// TIA Portal V17 export
// export: Created 2025-03-05T08:03:15.303072Z, ExportSetting WithDefaults, DisplayName Totally Integrated Automation Portal, DisplayVersion V17 Update 8, DisplayName TIA Portal Openness, DisplayVersion V17 Update 8, DisplayName TIA Portal Version Control Interface, DisplayVersion V17, DisplayName SINAMICS Startdrive Advanced, DisplayVersion V17 SP2, DisplayName SINAMICS Startdrive G110M, G120, G120C, G120D, G120P, G115D, DisplayVersion V17 SP2, DisplayName SINAMICS Startdrive G130, G150, S120, S150, SINAMICS MV, S210, DisplayVersion V17 SP2, DisplayName STEP 7 Professional, DisplayVersion V17 Update 8, DisplayName SINUMERIK ONE STEP 7 Toolbox, DisplayVersion V17 Update 12, DisplayName SINUMERIK 840D sl STEP 7 Toolbox, DisplayVersion V17 Update 12, DisplayName STEP 7 Safety, DisplayVersion V17 Update 6, DisplayName WinCC Advanced, DisplayVersion V17 Update 8
FUNCTION_BLOCK "FB22502_STIRRER_CONTROL"   // FB22502, LAD
{ S7_Optimized_Access := 'FALSE' }
VERSION : 0.1
// stored: AutoNumber false, IsIECCheckEnabled false, SetENOAutomatically false, UDAEnableTagReadback false
   VAR_INPUT
      CONTROL_ON_DELAYED : Bool;   // Control On Delayed
      MOTOR_CONDITIONS : Bool;   // Motor Conditions
      MOTOR_STATUS_ERROR : Bool;   // Motor Status Error
      MOTOR_STATUS_ENABLE : Bool;   // Motor Status Enable
      MOTOR_STATUS_REACHED : Bool;   // Motor Status Reached
      START_MANUAL_REQUEST : Bool;   // Start Manual Request
      START_SEMI_REQUEST : Bool;   // Start Semi Request
      START_AUTO_REQUEST : Bool;   // Start Auto Request
      START_PROGRAM_REQUEST : Bool;   // Start Program Request
      STOP_MANUAL_REQUEST : Bool;   // Stop Manual Request
      STOP_SEMI_REQUEST : Bool;   // Stop Semi Request
      STOP_AUTO_REQUEST : Bool;   // Stop Auto Request
      STOP_PROGRAM_REQUEST : Bool;   // Stop Program Request
      MOTOR_ACTUAL_POSITION : DInt;   // Motor Actual Position
      MOTOR_ACTUAL_VELOCITY : DInt;   // Motor Actual Velocity
      MOTOR_ACTUAL_CURRENT : DInt;   // Motor Actual Current
      MOTOR_ACTUAL_CURRENT_FILTERED : DInt;   // Motor Actual Current Filtered
      MOTOR_ACTUAL_TEMPERATURE : Real;   // Motor Actual Temperature
      MOTOR_STATUS_REGISTER : UDInt;   // Motor Status Register
   END_VAR
   VAR_OUTPUT
      "MOTOR _VELOCITY _TARGET _SOURCE" : DInt;   // MOTOR VELOCITY TARGET SOURCE
      "MOTOR _MODE _OF _OPERATION" : Int;   // MOTOR MODE OF OPERATION
      "MOTOR _ENABLE _POWER _STAGE" : Int;   // MOTOR ENABLE POWER STAGE
      "MOTOR _OUT1" : Bool;   // MOTOR OUT1
      "MOTOR _OUT2" : Bool;   // MOTOR OUT2
      "MOTOR _OUT3" : Bool;   // MOTOR OUT3
      "MOTOR _ENABLE _1" : Bool;   // MOTOR ENABLE 1
      "MOTOR _ENABLE _2" : Bool;   // MOTOR ENABLE 2
      "CURRENT _LIMIT _ALARM" : Bool;   // CURRENT LIMIT ALARM
      "TEMPRETATURE _LIMIT _ALARM" : Bool;   // TEMPRETATURE LIMIT ALARM
   END_VAR
   VAR DB_SPECIFIC
      DATA_STANDARD : "GENERAL_DATA_START_STOP";
      DATA_HMI : "HMI_DATA_START_STOP";
      INPUT_SETTINGS : Struct
         UNIT_NUMBER : Int;
         HOPPER_NUMBER : Int;
      END_STRUCT;
      ALARM_SETTINGS : Struct
         CURRENT_LIMIT : DInt;   // CURRENT LIMIT
         TEMPERATURE_LIMIT : Real;   // TEMPERATURE LIMIT
         TIMER_CURRENT_LIMIT : TON_TIME;   // TIMER CURRENT LIMIT
         TIMER_TEMPERATURE_LIMIT : TON_TIME;
      END_STRUCT;
      "HMI _SETPOINT _VELOCITY" : DInt;   // HMI SETPOINT VELOCITY
      "HMI _ACTUAL _POSITION" : DInt;   // HMI ACTUAL POSITION
      "HMI _ACTUAL _VELOCITY" : DInt;   // HMI ACTUAL VELOCITY
      "HMI _ACTUAL _CURRENT" : DInt;   // HMI ACTUAL CURRENT
      "HMI _ACTUAL _CURRENT _FILTERED" : DInt;   // HMI ACTUAL CURRENT FILTERED
      "HMI _STIRRER _LOW _RANGE" : DInt;   // HMI STIRRER LOW RANGE
      "HMI _STIRRER _HIGH _RANGE" : DInt;   // HMI STIRRER HIGH RANGE
      "PROGRAM _SETPOINT _VELOCITY" : DInt;   // PROGRAM SETPOINT VELOCITY
      "SETPOINT _VELOCITY" : DInt;   // SETPOINT VELOCITY
      "FEEDBACK _POSITION" : DInt;   // FEEDBACK POSITION
      "FEEDBACK _VELOCITY" : DInt;   // FEEDBACK VELOCITY
      "FEEDBACK _CURRENT" : DInt;   // FEEDBACK CURRENT
      "FEEDBACK _CURRENT _FILTERED" : DInt;   // FEEDBACK CURRENT FILTERED
      "FEEDBACK _TEMPERATURE" : Real;   // FEEDBACK TEMPERATURE
   END_VAR
   VAR_TEMP
      DB_NUMBER : DInt;
      RETVAL : Int;
   END_VAR
   // ALARM_SETTINGS.TIMER_CURRENT_LIMIT.PT := T#1s;
   // ALARM_SETTINGS.TIMER_TEMPERATURE_LIMIT.PT := T#1s;
   VAR_TEMP   // added for the SCL form of the ladder/FBD networks
      _w1 : Bool;
      _w2 : Bool;
   END_VAR
BEGIN

NETWORK
TITLE = READ INSTANCE DB NUMBER
      L     DINO;
      +     10#800000;
      T     #DB_NUMBER;


REGION Network 2: INPUTS
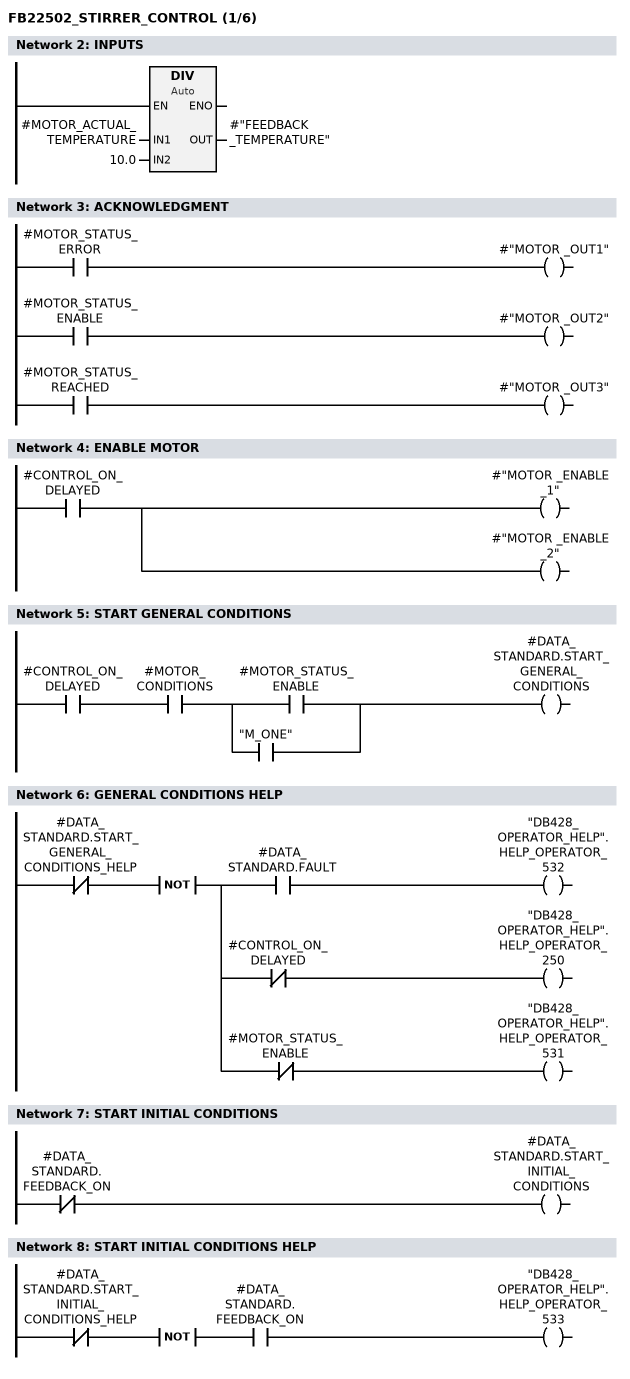
   RUNG wire#powerrail
      Div(in1 := #MOTOR_ACTUAL_TEMPERATURE, in2 := 10.0, out => #"FEEDBACK _TEMPERATURE")
   END_RUNG
   // the same network as SCL:
   #"FEEDBACK _TEMPERATURE" := #MOTOR_ACTUAL_TEMPERATURE / 10.0;
END_REGION

REGION Network 3: ACKNOWLEDGMENT
   RUNG wire#powerrail
      Contact( #MOTOR_STATUS_ERROR )
      Coil( #"MOTOR _OUT1" )
   END_RUNG
   RUNG wire#powerrail
      Contact( #MOTOR_STATUS_ENABLE )
      Coil( #"MOTOR _OUT2" )
   END_RUNG
   RUNG wire#powerrail
      Contact( #MOTOR_STATUS_REACHED )
      Coil( #"MOTOR _OUT3" )
   END_RUNG
   // the same network as SCL:
   #"MOTOR _OUT1" := #MOTOR_STATUS_ERROR;
   #"MOTOR _OUT2" := #MOTOR_STATUS_ENABLE;
   #"MOTOR _OUT3" := #MOTOR_STATUS_REACHED;
END_REGION

REGION Network 4: ENABLE MOTOR
   RUNG wire#powerrail
      Contact( #CONTROL_ON_DELAYED )
      wire#w1
      Coil( #"MOTOR _ENABLE _1" )
   END_RUNG
   RUNG wire#w1
      Coil( #"MOTOR _ENABLE _2" )
   END_RUNG
   // the same network as SCL:
   #"MOTOR _ENABLE _1" := #CONTROL_ON_DELAYED;
   #"MOTOR _ENABLE _2" := #CONTROL_ON_DELAYED;
END_REGION

REGION Network 5: START GENERAL CONDITIONS
   RUNG wire#powerrail
      Contact( #CONTROL_ON_DELAYED )
      Contact( #MOTOR_CONDITIONS )
      wire#w1
      Contact( #MOTOR_STATUS_ENABLE )
      wire#w2
      Coil( #DATA_STANDARD.START_GENERAL_CONDITIONS )
   END_RUNG
   RUNG wire#w1
      Contact( "M_ONE" )
   END_RUNG wire#w2
   // the same network as SCL:
   #DATA_STANDARD.START_GENERAL_CONDITIONS := #CONTROL_ON_DELAYED AND #MOTOR_CONDITIONS AND (#MOTOR_STATUS_ENABLE OR "M_ONE");
END_REGION

REGION Network 6: GENERAL CONDITIONS HELP
   RUNG wire#powerrail
      I_Contact( #DATA_STANDARD.START_GENERAL_CONDITIONS_HELP )
      Not()
      wire#w1
      Contact( #DATA_STANDARD.FAULT )
      Coil( "DB428_OPERATOR_HELP".HELP_OPERATOR_532 )
   END_RUNG
   RUNG wire#w1
      I_Contact( #CONTROL_ON_DELAYED )
      Coil( "DB428_OPERATOR_HELP".HELP_OPERATOR_250 )
   END_RUNG
   RUNG wire#w1
      I_Contact( #MOTOR_STATUS_ENABLE )
      Coil( "DB428_OPERATOR_HELP".HELP_OPERATOR_531 )
   END_RUNG
   // the same network as SCL:
   #_w1 := NOT (NOT #DATA_STANDARD.START_GENERAL_CONDITIONS_HELP);
   "DB428_OPERATOR_HELP".HELP_OPERATOR_532 := #_w1 AND #DATA_STANDARD.FAULT;
   "DB428_OPERATOR_HELP".HELP_OPERATOR_250 := #_w1 AND NOT #CONTROL_ON_DELAYED;
   "DB428_OPERATOR_HELP".HELP_OPERATOR_531 := #_w1 AND NOT #MOTOR_STATUS_ENABLE;
END_REGION

REGION Network 7: START INITIAL CONDITIONS
   RUNG wire#powerrail
      I_Contact( #DATA_STANDARD.FEEDBACK_ON )
      Coil( #DATA_STANDARD.START_INITIAL_CONDITIONS )
   END_RUNG
   // the same network as SCL:
   #DATA_STANDARD.START_INITIAL_CONDITIONS := NOT #DATA_STANDARD.FEEDBACK_ON;
END_REGION

REGION Network 8: START INITIAL CONDITIONS HELP
   RUNG wire#powerrail
      I_Contact( #DATA_STANDARD.START_INITIAL_CONDITIONS_HELP )
      Not()
      Contact( #DATA_STANDARD.FEEDBACK_ON )
      Coil( "DB428_OPERATOR_HELP".HELP_OPERATOR_533 )
   END_RUNG
   // the same network as SCL:
   "DB428_OPERATOR_HELP".HELP_OPERATOR_533 := NOT (NOT #DATA_STANDARD.START_INITIAL_CONDITIONS_HELP) AND #DATA_STANDARD.FEEDBACK_ON;
END_REGION

REGION Network 9: START MANUAL REQUEST
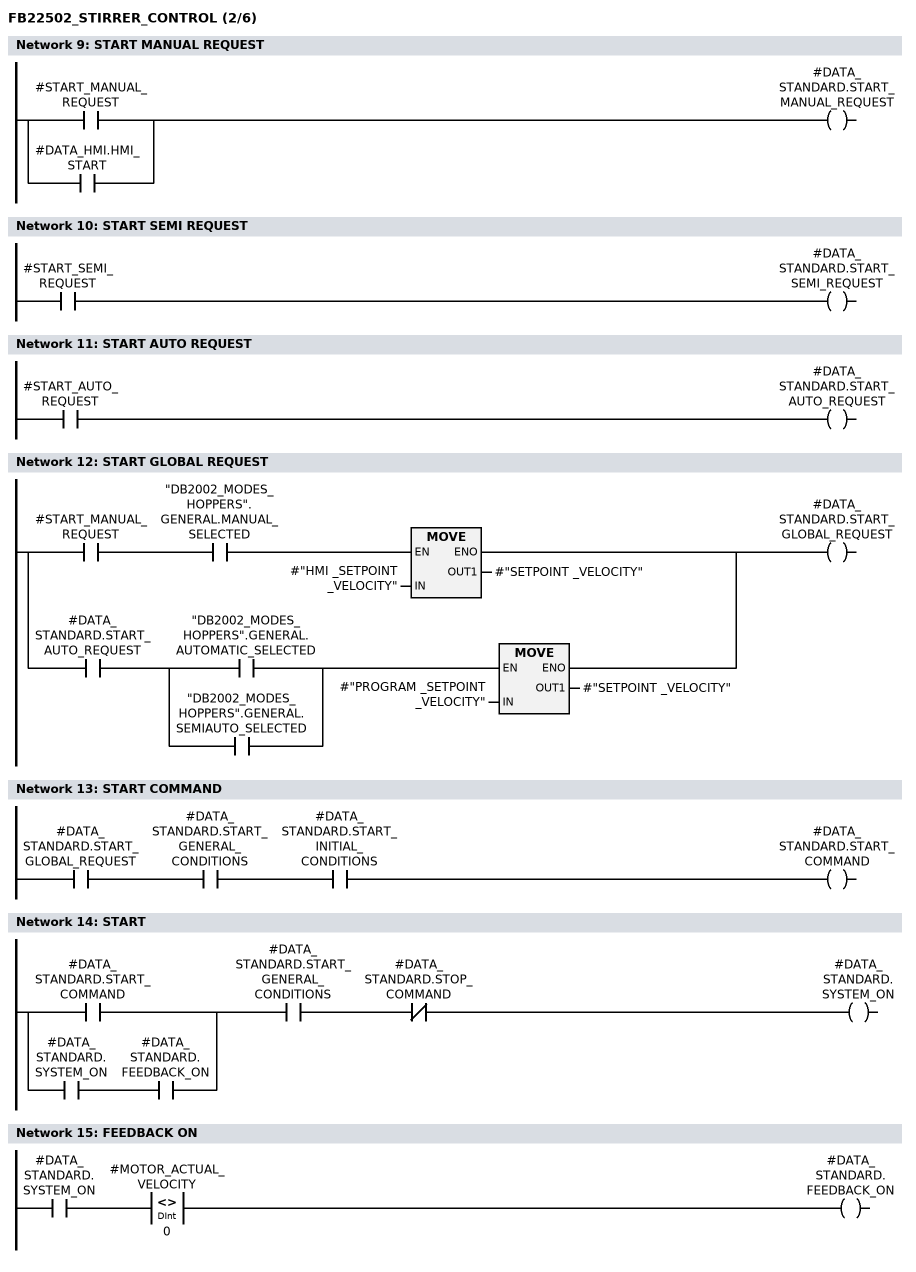
   RUNG wire#powerrail
      Contact( #START_MANUAL_REQUEST )
      wire#w1
      Coil( #DATA_STANDARD.START_MANUAL_REQUEST )
   END_RUNG
   RUNG wire#powerrail
      Contact( #DATA_HMI.HMI_START )
   END_RUNG wire#w1
   // the same network as SCL:
   #DATA_STANDARD.START_MANUAL_REQUEST := #START_MANUAL_REQUEST OR #DATA_HMI.HMI_START;
END_REGION

REGION Network 10: START SEMI REQUEST
   RUNG wire#powerrail
      Contact( #START_SEMI_REQUEST )
      Coil( #DATA_STANDARD.START_SEMI_REQUEST )
   END_RUNG
   // the same network as SCL:
   #DATA_STANDARD.START_SEMI_REQUEST := #START_SEMI_REQUEST;
END_REGION

REGION Network 11: START AUTO REQUEST
   RUNG wire#powerrail
      Contact( #START_AUTO_REQUEST )
      Coil( #DATA_STANDARD.START_AUTO_REQUEST )
   END_RUNG
   // the same network as SCL:
   #DATA_STANDARD.START_AUTO_REQUEST := #START_AUTO_REQUEST;
END_REGION

REGION Network 12: START GLOBAL REQUEST
   RUNG wire#powerrail
      Contact( #START_MANUAL_REQUEST )
      Contact( "DB2002_MODES_HOPPERS".GENERAL.MANUAL_SELECTED )
      Move(in := #"HMI _SETPOINT _VELOCITY", out1 => #"SETPOINT _VELOCITY")
      wire#w1
      Coil( #DATA_STANDARD.START_GLOBAL_REQUEST )
   END_RUNG
   RUNG wire#powerrail
      Contact( #DATA_STANDARD.START_AUTO_REQUEST )
      wire#w2
      Contact( "DB2002_MODES_HOPPERS".GENERAL.AUTOMATIC_SELECTED )
      wire#w3
      Move(in := #"PROGRAM _SETPOINT _VELOCITY", out1 => #"SETPOINT _VELOCITY")
   END_RUNG wire#w1
   RUNG wire#w2
      Contact( "DB2002_MODES_HOPPERS".GENERAL.SEMIAUTO_SELECTED )
   END_RUNG wire#w3
   // the same network as SCL:
   #_w1 := #START_MANUAL_REQUEST AND "DB2002_MODES_HOPPERS".GENERAL.MANUAL_SELECTED;
   IF #_w1 THEN #"SETPOINT _VELOCITY" := #"HMI _SETPOINT _VELOCITY"; END_IF;
   #_w2 := #DATA_STANDARD.START_AUTO_REQUEST AND ("DB2002_MODES_HOPPERS".GENERAL.AUTOMATIC_SELECTED OR "DB2002_MODES_HOPPERS".GENERAL.SEMIAUTO_SELECTED);
   IF #_w2 THEN #"SETPOINT _VELOCITY" := #"PROGRAM _SETPOINT _VELOCITY"; END_IF;
   #DATA_STANDARD.START_GLOBAL_REQUEST := #_w1 OR #_w2;
END_REGION

REGION Network 13: START COMMAND
   RUNG wire#powerrail
      Contact( #DATA_STANDARD.START_GLOBAL_REQUEST )
      Contact( #DATA_STANDARD.START_GENERAL_CONDITIONS )
      Contact( #DATA_STANDARD.START_INITIAL_CONDITIONS )
      Coil( #DATA_STANDARD.START_COMMAND )
   END_RUNG
   // the same network as SCL:
   #DATA_STANDARD.START_COMMAND := #DATA_STANDARD.START_GLOBAL_REQUEST AND #DATA_STANDARD.START_GENERAL_CONDITIONS AND #DATA_STANDARD.START_INITIAL_CONDITIONS;
END_REGION

REGION Network 14: START
   RUNG wire#powerrail
      Contact( #DATA_STANDARD.START_COMMAND )
      wire#w1
      Contact( #DATA_STANDARD.START_GENERAL_CONDITIONS )
      I_Contact( #DATA_STANDARD.STOP_COMMAND )
      Coil( #DATA_STANDARD.SYSTEM_ON )
   END_RUNG
   RUNG wire#powerrail
      Contact( #DATA_STANDARD.SYSTEM_ON )
      Contact( #DATA_STANDARD.FEEDBACK_ON )
   END_RUNG wire#w1
   // the same network as SCL:
   #DATA_STANDARD.SYSTEM_ON := (#DATA_STANDARD.START_COMMAND OR (#DATA_STANDARD.SYSTEM_ON AND #DATA_STANDARD.FEEDBACK_ON)) AND #DATA_STANDARD.START_GENERAL_CONDITIONS AND NOT #DATA_STANDARD.STOP_COMMAND;
END_REGION

REGION Network 15: FEEDBACK ON
   RUNG wire#powerrail
      Contact( #DATA_STANDARD.SYSTEM_ON )
      { S7_Templates := "SrcType := DInt" } NE_Contact(in1 := #MOTOR_ACTUAL_VELOCITY, in2 := 0)
      Coil( #DATA_STANDARD.FEEDBACK_ON )
   END_RUNG
   // the same network as SCL:
   #DATA_STANDARD.FEEDBACK_ON := #DATA_STANDARD.SYSTEM_ON AND (#MOTOR_ACTUAL_VELOCITY <> 0);
END_REGION

REGION Network 16: STOP GENERAL CONDITIONS
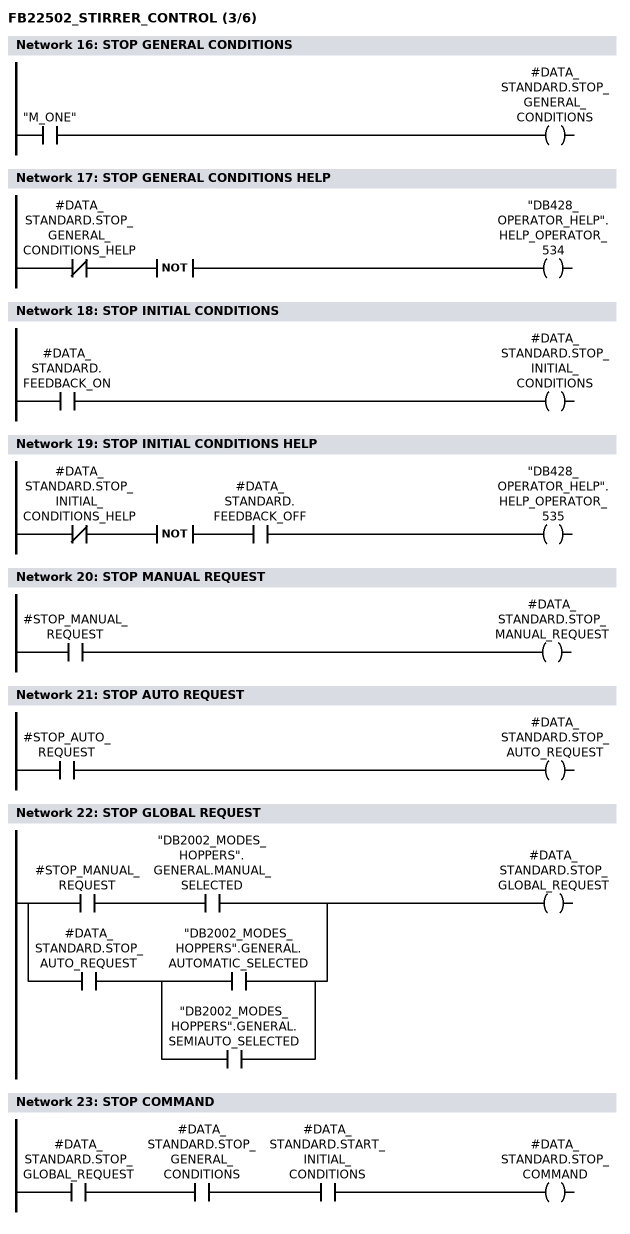
   RUNG wire#powerrail
      Contact( "M_ONE" )
      Coil( #DATA_STANDARD.STOP_GENERAL_CONDITIONS )
   END_RUNG
   // the same network as SCL:
   #DATA_STANDARD.STOP_GENERAL_CONDITIONS := "M_ONE";
END_REGION

REGION Network 17: STOP GENERAL CONDITIONS HELP
   RUNG wire#powerrail
      I_Contact( #DATA_STANDARD.STOP_GENERAL_CONDITIONS_HELP )
      Not()
      Coil( "DB428_OPERATOR_HELP".HELP_OPERATOR_534 )
   END_RUNG
   // the same network as SCL:
   "DB428_OPERATOR_HELP".HELP_OPERATOR_534 := NOT (NOT #DATA_STANDARD.STOP_GENERAL_CONDITIONS_HELP);
END_REGION

REGION Network 18: STOP INITIAL CONDITIONS
   RUNG wire#powerrail
      Contact( #DATA_STANDARD.FEEDBACK_ON )
      Coil( #DATA_STANDARD.STOP_INITIAL_CONDITIONS )
   END_RUNG
   // the same network as SCL:
   #DATA_STANDARD.STOP_INITIAL_CONDITIONS := #DATA_STANDARD.FEEDBACK_ON;
END_REGION

REGION Network 19: STOP INITIAL CONDITIONS HELP
   RUNG wire#powerrail
      I_Contact( #DATA_STANDARD.STOP_INITIAL_CONDITIONS_HELP )
      Not()
      Contact( #DATA_STANDARD.FEEDBACK_OFF )
      Coil( "DB428_OPERATOR_HELP".HELP_OPERATOR_535 )
   END_RUNG
   // the same network as SCL:
   "DB428_OPERATOR_HELP".HELP_OPERATOR_535 := NOT (NOT #DATA_STANDARD.STOP_INITIAL_CONDITIONS_HELP) AND #DATA_STANDARD.FEEDBACK_OFF;
END_REGION

REGION Network 20: STOP MANUAL REQUEST
   RUNG wire#powerrail
      Contact( #STOP_MANUAL_REQUEST )
      Coil( #DATA_STANDARD.STOP_MANUAL_REQUEST )
   END_RUNG
   // the same network as SCL:
   #DATA_STANDARD.STOP_MANUAL_REQUEST := #STOP_MANUAL_REQUEST;
END_REGION

REGION Network 21: STOP AUTO REQUEST
   RUNG wire#powerrail
      Contact( #STOP_AUTO_REQUEST )
      Coil( #DATA_STANDARD.STOP_AUTO_REQUEST )
   END_RUNG
   // the same network as SCL:
   #DATA_STANDARD.STOP_AUTO_REQUEST := #STOP_AUTO_REQUEST;
END_REGION

REGION Network 22: STOP GLOBAL REQUEST
   RUNG wire#powerrail
      Contact( #STOP_MANUAL_REQUEST )
      Contact( "DB2002_MODES_HOPPERS".GENERAL.MANUAL_SELECTED )
      wire#w1
      Coil( #DATA_STANDARD.STOP_GLOBAL_REQUEST )
   END_RUNG
   RUNG wire#powerrail
      Contact( #DATA_STANDARD.STOP_AUTO_REQUEST )
      wire#w2
      Contact( "DB2002_MODES_HOPPERS".GENERAL.AUTOMATIC_SELECTED )
   END_RUNG wire#w1
   RUNG wire#w2
      Contact( "DB2002_MODES_HOPPERS".GENERAL.SEMIAUTO_SELECTED )
   END_RUNG wire#w1
   // the same network as SCL:
   #DATA_STANDARD.STOP_GLOBAL_REQUEST := (#STOP_MANUAL_REQUEST AND "DB2002_MODES_HOPPERS".GENERAL.MANUAL_SELECTED) OR (#DATA_STANDARD.STOP_AUTO_REQUEST AND ("DB2002_MODES_HOPPERS".GENERAL.AUTOMATIC_SELECTED OR "DB2002_MODES_HOPPERS".GENERAL.SEMIAUTO_SELECTED));
END_REGION

REGION Network 23: STOP COMMAND
   RUNG wire#powerrail
      Contact( #DATA_STANDARD.STOP_GLOBAL_REQUEST )
      Contact( #DATA_STANDARD.STOP_GENERAL_CONDITIONS )
      Contact( #DATA_STANDARD.START_INITIAL_CONDITIONS )
      Coil( #DATA_STANDARD.STOP_COMMAND )
   END_RUNG
   // the same network as SCL:
   #DATA_STANDARD.STOP_COMMAND := #DATA_STANDARD.STOP_GLOBAL_REQUEST AND #DATA_STANDARD.STOP_GENERAL_CONDITIONS AND #DATA_STANDARD.START_INITIAL_CONDITIONS;
END_REGION

REGION Network 24: STOP
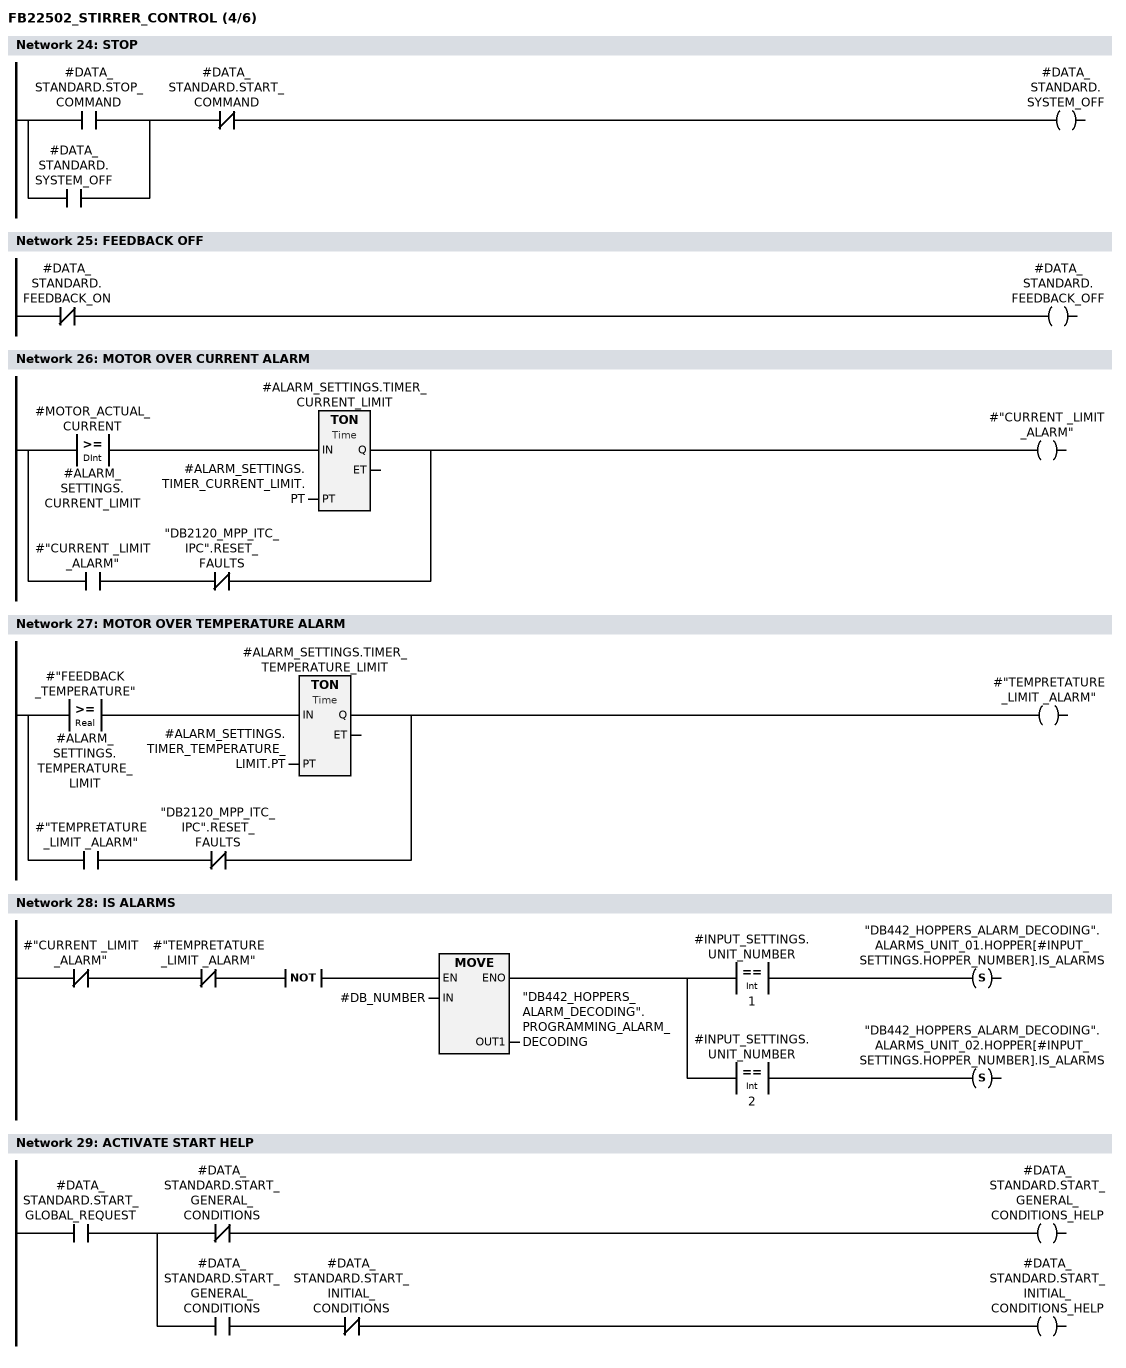
   RUNG wire#powerrail
      Contact( #DATA_STANDARD.STOP_COMMAND )
      wire#w1
      I_Contact( #DATA_STANDARD.START_COMMAND )
      Coil( #DATA_STANDARD.SYSTEM_OFF )
   END_RUNG
   RUNG wire#powerrail
      Contact( #DATA_STANDARD.SYSTEM_OFF )
   END_RUNG wire#w1
   // the same network as SCL:
   #DATA_STANDARD.SYSTEM_OFF := (#DATA_STANDARD.STOP_COMMAND OR #DATA_STANDARD.SYSTEM_OFF) AND NOT #DATA_STANDARD.START_COMMAND;
END_REGION

REGION Network 25: FEEDBACK OFF
   RUNG wire#powerrail
      I_Contact( #DATA_STANDARD.FEEDBACK_ON )
      Coil( #DATA_STANDARD.FEEDBACK_OFF )
   END_RUNG
   // the same network as SCL:
   #DATA_STANDARD.FEEDBACK_OFF := NOT #DATA_STANDARD.FEEDBACK_ON;
END_REGION

REGION Network 26: MOTOR OVER CURRENT ALARM
   RUNG wire#powerrail
      { S7_Templates := "SrcType := DInt" } GE_Contact(in1 := #MOTOR_ACTUAL_CURRENT, in2 := #ALARM_SETTINGS.CURRENT_LIMIT)
      { S7_Templates := "time_type := Time" } #ALARM_SETTINGS.TIMER_CURRENT_LIMIT.TON(pt := #ALARM_SETTINGS.TIMER_CURRENT_LIMIT.PT, et =>)
      wire#w1
      Coil( #"CURRENT _LIMIT _ALARM" )
   END_RUNG
   RUNG wire#powerrail
      Contact( #"CURRENT _LIMIT _ALARM" )
      I_Contact( "DB2120_MPP_ITC_IPC".RESET_FAULTS )
   END_RUNG wire#w1
   // the same network as SCL:
   #ALARM_SETTINGS.TIMER_CURRENT_LIMIT.TON(IN := #MOTOR_ACTUAL_CURRENT >= #ALARM_SETTINGS.CURRENT_LIMIT,
                           PT := #ALARM_SETTINGS.TIMER_CURRENT_LIMIT.PT);
   #"CURRENT _LIMIT _ALARM" := #ALARM_SETTINGS.TIMER_CURRENT_LIMIT.Q OR (#"CURRENT _LIMIT _ALARM" AND NOT "DB2120_MPP_ITC_IPC".RESET_FAULTS);
END_REGION

REGION Network 27: MOTOR OVER TEMPERATURE ALARM
   RUNG wire#powerrail
      { S7_Templates := "SrcType := Real" } GE_Contact(in1 := #"FEEDBACK _TEMPERATURE", in2 := #ALARM_SETTINGS.TEMPERATURE_LIMIT)
      { S7_Templates := "time_type := Time" } #ALARM_SETTINGS.TIMER_TEMPERATURE_LIMIT.TON(pt := #ALARM_SETTINGS.TIMER_TEMPERATURE_LIMIT.PT, et =>)
      wire#w1
      Coil( #"TEMPRETATURE _LIMIT _ALARM" )
   END_RUNG
   RUNG wire#powerrail
      Contact( #"TEMPRETATURE _LIMIT _ALARM" )
      I_Contact( "DB2120_MPP_ITC_IPC".RESET_FAULTS )
   END_RUNG wire#w1
   // the same network as SCL:
   #ALARM_SETTINGS.TIMER_TEMPERATURE_LIMIT.TON(IN := #"FEEDBACK _TEMPERATURE" >= #ALARM_SETTINGS.TEMPERATURE_LIMIT,
                           PT := #ALARM_SETTINGS.TIMER_TEMPERATURE_LIMIT.PT);
   #"TEMPRETATURE _LIMIT _ALARM" := #ALARM_SETTINGS.TIMER_TEMPERATURE_LIMIT.Q OR (#"TEMPRETATURE _LIMIT _ALARM" AND NOT "DB2120_MPP_ITC_IPC".RESET_FAULTS);
END_REGION

REGION Network 28: IS ALARMS
   RUNG wire#powerrail
      I_Contact( #"CURRENT _LIMIT _ALARM" )
      I_Contact( #"TEMPRETATURE _LIMIT _ALARM" )
      Not()
      Move(in := #DB_NUMBER, out1 => "DB442_HOPPERS_ALARM_DECODING".PROGRAMMING_ALARM_DECODING)
      wire#w1
      { S7_Templates := "SrcType := Int" } EQ_Contact(in1 := #INPUT_SETTINGS.UNIT_NUMBER, in2 := 1)
      S_Coil( "DB442_HOPPERS_ALARM_DECODING".ALARMS_UNIT_01.HOPPER[#INPUT_SETTINGS.HOPPER_NUMBER].IS_ALARMS )
   END_RUNG
   RUNG wire#w1
      { S7_Templates := "SrcType := Int" } EQ_Contact(in1 := #INPUT_SETTINGS.UNIT_NUMBER, in2 := 2)
      S_Coil( "DB442_HOPPERS_ALARM_DECODING".ALARMS_UNIT_02.HOPPER[#INPUT_SETTINGS.HOPPER_NUMBER].IS_ALARMS )
   END_RUNG
   // the same network as SCL:
   #_w1 := NOT (NOT #"CURRENT _LIMIT _ALARM" AND NOT #"TEMPRETATURE _LIMIT _ALARM");
   IF #_w1 THEN "DB442_HOPPERS_ALARM_DECODING".PROGRAMMING_ALARM_DECODING := #DB_NUMBER; END_IF;
   IF #_w1 AND (#INPUT_SETTINGS.UNIT_NUMBER = 1) THEN
       "DB442_HOPPERS_ALARM_DECODING".ALARMS_UNIT_01.HOPPER[#INPUT_SETTINGS.HOPPER_NUMBER].IS_ALARMS := TRUE;
   END_IF;
   IF #_w1 AND (#INPUT_SETTINGS.UNIT_NUMBER = 2) THEN
       "DB442_HOPPERS_ALARM_DECODING".ALARMS_UNIT_02.HOPPER[#INPUT_SETTINGS.HOPPER_NUMBER].IS_ALARMS := TRUE;
   END_IF;
END_REGION

REGION Network 29: ACTIVATE START HELP
   RUNG wire#powerrail
      Contact( #DATA_STANDARD.START_GLOBAL_REQUEST )
      wire#w1
      I_Contact( #DATA_STANDARD.START_GENERAL_CONDITIONS )
      Coil( #DATA_STANDARD.START_GENERAL_CONDITIONS_HELP )
   END_RUNG
   RUNG wire#w1
      Contact( #DATA_STANDARD.START_GENERAL_CONDITIONS )
      I_Contact( #DATA_STANDARD.START_INITIAL_CONDITIONS )
      Coil( #DATA_STANDARD.START_INITIAL_CONDITIONS_HELP )
   END_RUNG
   // the same network as SCL:
   #DATA_STANDARD.START_GENERAL_CONDITIONS_HELP := #DATA_STANDARD.START_GLOBAL_REQUEST AND NOT #DATA_STANDARD.START_GENERAL_CONDITIONS;
   #DATA_STANDARD.START_INITIAL_CONDITIONS_HELP := #DATA_STANDARD.START_GLOBAL_REQUEST AND #DATA_STANDARD.START_GENERAL_CONDITIONS AND NOT #DATA_STANDARD.START_INITIAL_CONDITIONS;
END_REGION

REGION Network 30: ACTIVATE STOP HELP
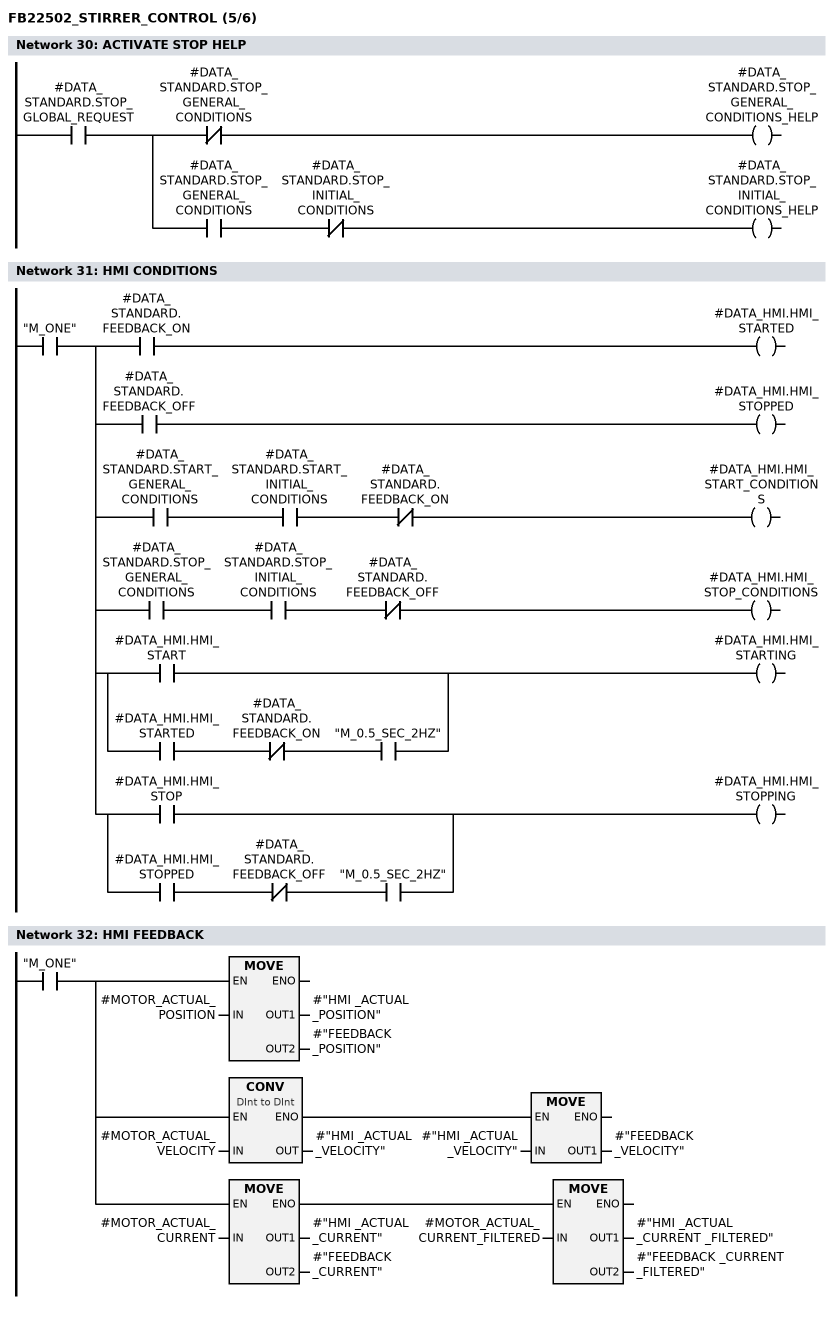
   RUNG wire#powerrail
      Contact( #DATA_STANDARD.STOP_GLOBAL_REQUEST )
      wire#w1
      I_Contact( #DATA_STANDARD.STOP_GENERAL_CONDITIONS )
      Coil( #DATA_STANDARD.STOP_GENERAL_CONDITIONS_HELP )
   END_RUNG
   RUNG wire#w1
      Contact( #DATA_STANDARD.STOP_GENERAL_CONDITIONS )
      I_Contact( #DATA_STANDARD.STOP_INITIAL_CONDITIONS )
      Coil( #DATA_STANDARD.STOP_INITIAL_CONDITIONS_HELP )
   END_RUNG
   // the same network as SCL:
   #DATA_STANDARD.STOP_GENERAL_CONDITIONS_HELP := #DATA_STANDARD.STOP_GLOBAL_REQUEST AND NOT #DATA_STANDARD.STOP_GENERAL_CONDITIONS;
   #DATA_STANDARD.STOP_INITIAL_CONDITIONS_HELP := #DATA_STANDARD.STOP_GLOBAL_REQUEST AND #DATA_STANDARD.STOP_GENERAL_CONDITIONS AND NOT #DATA_STANDARD.STOP_INITIAL_CONDITIONS;
END_REGION

REGION Network 31: HMI CONDITIONS
   RUNG wire#powerrail
      Contact( "M_ONE" )
      wire#w1
      Contact( #DATA_STANDARD.FEEDBACK_ON )
      Coil( #DATA_HMI.HMI_STARTED )
   END_RUNG
   RUNG wire#w1
      Contact( #DATA_STANDARD.FEEDBACK_OFF )
      Coil( #DATA_HMI.HMI_STOPPED )
   END_RUNG
   RUNG wire#w1
      Contact( #DATA_STANDARD.START_GENERAL_CONDITIONS )
      Contact( #DATA_STANDARD.START_INITIAL_CONDITIONS )
      I_Contact( #DATA_STANDARD.FEEDBACK_ON )
      Coil( #DATA_HMI.HMI_START_CONDITIONS )
   END_RUNG
   RUNG wire#w1
      Contact( #DATA_STANDARD.STOP_GENERAL_CONDITIONS )
      Contact( #DATA_STANDARD.STOP_INITIAL_CONDITIONS )
      I_Contact( #DATA_STANDARD.FEEDBACK_OFF )
      Coil( #DATA_HMI.HMI_STOP_CONDITIONS )
   END_RUNG
   RUNG wire#w1
      Contact( #DATA_HMI.HMI_START )
      wire#w2
      Coil( #DATA_HMI.HMI_STARTING )
   END_RUNG
   RUNG wire#w1
      Contact( #DATA_HMI.HMI_STARTED )
      I_Contact( #DATA_STANDARD.FEEDBACK_ON )
      Contact( "M_0.5_SEC_2HZ" )
   END_RUNG wire#w2
   RUNG wire#w1
      Contact( #DATA_HMI.HMI_STOP )
      wire#w3
      Coil( #DATA_HMI.HMI_STOPPING )
   END_RUNG
   RUNG wire#w1
      Contact( #DATA_HMI.HMI_STOPPED )
      I_Contact( #DATA_STANDARD.FEEDBACK_OFF )
      Contact( "M_0.5_SEC_2HZ" )
   END_RUNG wire#w3
   // the same network as SCL:
   #DATA_HMI.HMI_STARTED := "M_ONE" AND #DATA_STANDARD.FEEDBACK_ON;
   #DATA_HMI.HMI_STOPPED := "M_ONE" AND #DATA_STANDARD.FEEDBACK_OFF;
   #DATA_HMI.HMI_START_CONDITIONS := "M_ONE" AND #DATA_STANDARD.START_GENERAL_CONDITIONS AND #DATA_STANDARD.START_INITIAL_CONDITIONS AND NOT #DATA_STANDARD.FEEDBACK_ON;
   #DATA_HMI.HMI_STOP_CONDITIONS := "M_ONE" AND #DATA_STANDARD.STOP_GENERAL_CONDITIONS AND #DATA_STANDARD.STOP_INITIAL_CONDITIONS AND NOT #DATA_STANDARD.FEEDBACK_OFF;
   #DATA_HMI.HMI_STARTING := "M_ONE" AND (#DATA_HMI.HMI_START OR (#DATA_HMI.HMI_STARTED AND NOT #DATA_STANDARD.FEEDBACK_ON AND "M_0.5_SEC_2HZ"));
   #DATA_HMI.HMI_STOPPING := "M_ONE" AND (#DATA_HMI.HMI_STOP OR (#DATA_HMI.HMI_STOPPED AND NOT #DATA_STANDARD.FEEDBACK_OFF AND "M_0.5_SEC_2HZ"));
END_REGION

REGION Network 32: HMI FEEDBACK
   RUNG wire#powerrail
      Contact( "M_ONE" )
      wire#w1
      Move(in := #MOTOR_ACTUAL_POSITION, out1 => #"HMI _ACTUAL _POSITION", out2 => #"FEEDBACK _POSITION")
   END_RUNG
   RUNG wire#w1
      { S7_Templates := "[SrcType := DInt, DestType := DInt]" } Convert(in := #MOTOR_ACTUAL_VELOCITY, out => #"HMI _ACTUAL _VELOCITY")
      Move(in := #"HMI _ACTUAL _VELOCITY", out1 => #"FEEDBACK _VELOCITY")
   END_RUNG
   RUNG wire#w1
      Move(in := #MOTOR_ACTUAL_CURRENT, out1 => #"HMI _ACTUAL _CURRENT", out2 => #"FEEDBACK _CURRENT")
      Move(in := #MOTOR_ACTUAL_CURRENT_FILTERED, out1 => #"HMI _ACTUAL _CURRENT _FILTERED", out2 => #"FEEDBACK _CURRENT _FILTERED")
   END_RUNG
   // the same network as SCL:
   IF "M_ONE" THEN
       #"HMI _ACTUAL _POSITION" := #MOTOR_ACTUAL_POSITION;
       #"FEEDBACK _POSITION" := #MOTOR_ACTUAL_POSITION;
       #"HMI _ACTUAL _VELOCITY" := DINT_TO_DINT(#MOTOR_ACTUAL_VELOCITY);
       #"FEEDBACK _VELOCITY" := #"HMI _ACTUAL _VELOCITY";
       #"HMI _ACTUAL _CURRENT" := #MOTOR_ACTUAL_CURRENT;
       #"FEEDBACK _CURRENT" := #MOTOR_ACTUAL_CURRENT;
       #"HMI _ACTUAL _CURRENT _FILTERED" := #MOTOR_ACTUAL_CURRENT_FILTERED;
       #"FEEDBACK _CURRENT _FILTERED" := #MOTOR_ACTUAL_CURRENT_FILTERED;
   END_IF;
END_REGION

REGION Network 33: OUTPUT
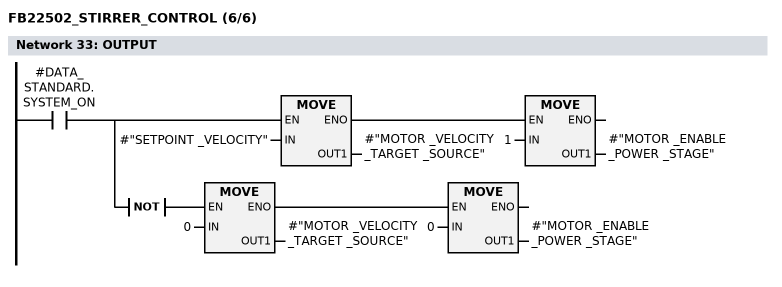
   RUNG wire#powerrail
      Contact( #DATA_STANDARD.SYSTEM_ON )
      wire#w1
      Move(in := #"SETPOINT _VELOCITY", out1 => #"MOTOR _VELOCITY _TARGET _SOURCE")
      Move(in := 1, out1 => #"MOTOR _ENABLE _POWER _STAGE")
   END_RUNG
   RUNG wire#w1
      Not()
      Move(in := 0, out1 => #"MOTOR _VELOCITY _TARGET _SOURCE")
      Move(in := 0, out1 => #"MOTOR _ENABLE _POWER _STAGE")
   END_RUNG
   // the same network as SCL:
   IF #DATA_STANDARD.SYSTEM_ON THEN
       #"MOTOR _VELOCITY _TARGET _SOURCE" := #"SETPOINT _VELOCITY";
       #"MOTOR _ENABLE _POWER _STAGE" := 1;
   END_IF;
   IF NOT #DATA_STANDARD.SYSTEM_ON THEN
       #"MOTOR _VELOCITY _TARGET _SOURCE" := 0;
       #"MOTOR _ENABLE _POWER _STAGE" := 0;
   END_IF;
END_REGION
END_FUNCTION_BLOCK
